Staubli VAL3: setResolution.pgx

public program setResolution(num x_nResolution)
begin
  // This routine sets the encoder resolution
  //
  // Input Param
  //    x_nEncResolution  : Encoder resolution.
  //
  // Output Param
  //    none
  //
  //----------------------------------------------------------------
  //
  if ioStatus(aoEncResolution)>=0
    aioSet(aoEncResolution,x_nResolution)
    nEncResolution=x_nResolution
  endIf
end
